# EPICS autosave request: specsAnalyserApp/Db/specsManipulator.req
$(P)$(R)MOVE
$(P)$(R)MOVE_RBV
$(P)$(R)DIRECT_MOVE
$(P)$(R)DIRECT_MOVE_RBV
